// TIA Portal V18 export
FUNCTION "IOupdate_General" : Void   // FC10000, LAD
{ S7_Optimized_Access := 'TRUE' }
VERSION : 0.1
// stored: AutoNumber false, IsIECCheckEnabled false, SetENOAutomatically false, UDAEnableTagReadback false
BEGIN

REGION Network 1
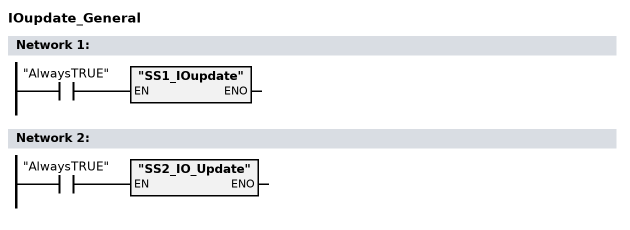
   RUNG wire#powerrail
      Contact( "AlwaysTRUE" )
      "SS1_IOupdate"()
   END_RUNG
   // the same network as SCL:
   IF "AlwaysTRUE" THEN "SS1_IOupdate"(); END_IF;
END_REGION

REGION Network 2
   RUNG wire#powerrail
      Contact( "AlwaysTRUE" )
      "SS2_IO_Update"()
   END_RUNG
   // the same network as SCL:
   IF "AlwaysTRUE" THEN "SS2_IO_Update"(); END_IF;
END_REGION
END_FUNCTION
